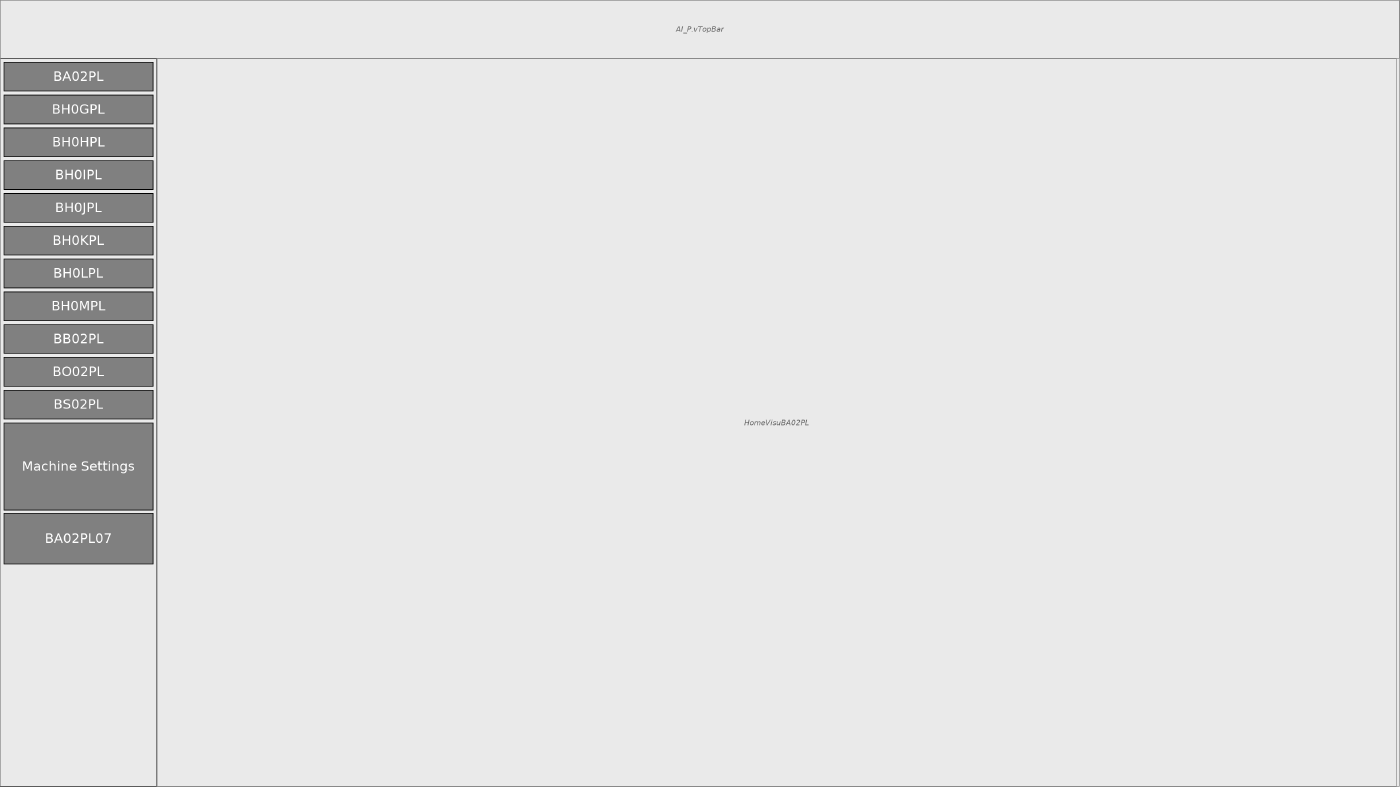
VISUALIZATION HomeVisu_1  // 1920x1080
    Rectangle (0,80 215x1000)
    Frame (215,80 1700x1000)
        shows HomeVisuBA02PL()
        shows HomeVisuBH0GPL()
        shows HomeVisuBH0HPL()
        shows HomeVisuBH0IPL()
        shows HomeVisuBH0JPL()
        shows HomeVisuBH0KPL()
        shows HomeVisuBH0LPL()
        shows HomeVisuBH0MPL()
        shows HomeVisuBB02PL()
        shows HomeVisuBO02PL()
        shows HomeVisuBS02PL()
        shows vHotPlateSettings_V3_B02PL(fbHP1_M1 := MAIN.fbHotPlate_G1_M1, fbHP1_M2 := MAIN.fbHotPlate_G1_M2, fbHP1_M3 := MAIN.fbHotPlate_G1_M3, fbHP2_M1 := MAIN.fbHotPlate_G2_M1, fbHP2_M2 := MAIN.fbHotPlate_G2_M2, fbHP2_M3 := MAIN.fbHotPlate_G2_M3, fbHP3_M1 := MAIN.fbHotPlate_G3_M1, fbHP3_M2 := MAIN.fbHotPlate_G3_M2, fbHP3_M3 := MAIN.fbHotPlate_G3_M3, fbHP4_M1 := MAIN.fbHotPlate_G4_M1, fbHP4_M2 := MAIN.fbHotPlate_G4_M2, fbHP4_M3 := MAIN.fbHotPlate_G4_M3, fbHP5_M1 := MAIN.fbHotPlate_G5_M1, fbHP5_M2 := MAIN.fbHotPlate_G5_M2, fbHP5_M3 := MAIN.fbHotPlate_G5_M3, fbHP6_M1 := MAIN.fbHotPlate_G6_M1, fbHP6_M2 := MAIN.fbHotPlate_G6_M2, fbHP6_M3 := MAIN.fbHotPlate_G6_M3, fbHP7_M1 := MAIN.fbHotPlate_G7_M1, fbHP7_M2 := MAIN.fbHotPlate_G7_M2, fbHP7_M3 := MAIN.fbHotPlate_G7_M3, fbS01_Press := MAIN.fbS01_BearingPress, fbS01_FixtureBase := MAIN.fbS01_KeyencePNVisSens, fbS02_Press := MAIN.fbS02_BearingPress, fbS03_Press := MAIN.fbS03_BearingPress, fbS03_FixtureBase := MAIN.fbS03_CapFixture, fbS04_Press := MAIN.fbS04_BearingPress, stHMIData_Filler_A := MAIN.fb_Filler_A_Machine.stHMI, stParams_Filler_A := MAIN.fb_Filler_A_Machine.stSlaveParms, stHMIData_Cork := MAIN.fb_Cork_Machine.stHMI, stParams_Cork := MAIN.fb_Cork_Machine.stSlaveParms, stHMIData_Filler_B := MAIN.fb_Filler_B_Machine.stHMI, stParams_Filler_B := MAIN.fb_Filler_B_Machine.stSlaveParms, stHMIData_Sticker := MAIN.fb_Sticker_Machine.stHMI, stParams_Sticker := MAIN.fb_Sticker_Machine.stSlaveParms, stHMIData_Laser := MAIN.fb_Laser_Machine.stHMI, stParams_Laser := MAIN.fb_Laser_Machine.stSlaveParms, stHMI_Laser := MAIN.fb_Laser_Machine.fbLaserControl.stHMI_Laser, fbSonic_S02 := MAIN.fb_1_SonicTech_SonictechUSW, fbSonic_S04 := MAIN.fb_2_SonicTech_SonictechUSW, fbVacuumChamber := MAIN.fb_UnderPressure_Tester_Machine, fbTransporter := MAIN.fbTransporterUnderpressure)
        shows AI_M.vWeighingTunnel(fbWeighingTunel := MAIN.fbWeighingTunel)
        shows vWeighingTunelVisionFrame()
        shows vStations19_21_22()
        p3043078949: MAIN.fbLL19_1_EOL3
        p1709583229: GVL.stLL19_EOL_Settings_I
        p2719655782: MAIN.fbLL19_2_EOL3
        p3094409976: GVL.stLL19_EOL_Settings_II
        p74549115: 'Left chamber'
        p3369830373: 'Right chamber'
        p4001053958: MAIN.fbS21_DetectionTunel
        p3623223747: MAIN.fbS21_DetectionTunel
        p3171485557: GVL.stS21_DTL_WorkParams
        p817651737: MAIN.stStation_LCA01PL_SCA01PL21
        p3449029454: GVL.stS21_DTL_Settings
        p3777340465: MAIN.fbS19_RecipeManager
        p3453682166: MAIN.stS19_EOL3_TMP_TestParams
        p3169997168: GVL_IO.stS21_DTL_InOuts.iLaserCurrentValue
        p2878062980: MAIN.fbS11_ResWelder.fbPIM
        p847417406: MAIN.fbS12_HiosScrewDriver.fbPIM
        p1166385320: MAIN.fbS13_FrontFanPress.fbPIM
        p3688969483: MAIN.fbS14_AssemblyPostCtrl.fbPIM
        p2900755869: MAIN.fbS15_AssemblyPostCtrl.fbPIM
        p3528948000: MAIN.fbS18_LabelSticking.fbPIM
        p514386723: MAIN.fbS22_SetPackingStation
        p2740858475: MAIN.fbS18_LabelSticking.stInOuts.iPressure
        p901175331: MAIN.fbS18_LabelSticking.stTestParams
        p1258792094: MAIN.fbS15_AssemblyPostCtrl.stWorkParams
        p1006670856: MAIN.fbS14_AssemblyPostCtrl.stWorkParams
        p2724463019: MAIN.fbS13_FrontFanPress.stParams
        p3580047677: MAIN.fbS12_HiosScrewDriver.stTestParam
        p1282039943: MAIN.fbS11_ResWelder.stWorkParams
        p285620971: GVL.stS19_EOL_TestParams
        p2487237938: MAIN.fbS19_1_EOL3
        p1850671185: MAIN.fbS19_2_EOL3
        p4100169850: GVL.stS19_EOL_Settings_I
        p241999129: GVL.stS19_EOL_Settings_II
        p1128139719: MAIN.fbS11_ResWelder.fbPIM
        p3661060733: MAIN.fbS12_HiosScrewDriver.fbPIM
        p2905631467: MAIN.fbS13_FrontFanPress.fbPIM
        p861208392: MAIN.fbS14_AssemblyPostCtrl.fbPIM
        p1146343390: MAIN.fbS15_AssemblyPostCtrl.fbPIM
        p987935587: MAIN.fbS18_LabelSticking.fbPIM
        p3446969237: GVL.stS18_ManometerCalibration_TestData
        p715956300: GVL.stS18_PressureScalingData
        p3016093480: GVL.stS15_AssemblyPostParams
        p3301105598: GVL.stS14_AssemblyPostParams
        p1520847389: GVL.stS13_Parameters
        p765557387: GVL.stS12_Parameters
        p3030919985: MAIN.fbS11_ResWelder.stWorkParams
        p4053094083: MAIN.fbS22_SetPackingStation
        p662549438: MAIN.fbS18_LabelSticking.stInOuts.iPressure
        p2928623001: GVL.stS18_PressureScalingData
        p1931357957: MAIN.fbS01_SonictechUSW.fbPIM
        p2635091497: MAIN.fbS03_SonictechUSW.fbPIM
        p1953753884: MAIN.fbS05_1_SonictechUSW.fbPIM
        p3984243366: MAIN.fbS06_SonictechUSW.fbPIM
        p2591918640: MAIN.fbS07_SonictechUSW.fbPIM
        p180524961: MAIN.fbS08_SonictechUSW.fbPIM
        p2110105399: MAIN.fbS09_SonictechUSW.fbPIM
        p486682322: MAIN.fbS10_SonictechUSW.fbPIM
        p4100033511: MAIN.fbS16_SonictechUSW.fbPIM
        p2204547953: MAIN.fbS17_SonictechUSW.fbPIM
        p3358502448: MAIN.fbS07_FixCarrierPistonAssy.stInOuts.rHeatStampTemperature
        p3363745968: GVL.stS01_FixSettings
        p644927900: GVL.stS03_FixSettings
        p3474158761: GVL.stS05_BallPressSettings
        p2347394456: GVL.stS05_USWelderSettings
        p1444554003: GVL.stS06_FixSettings
        p555554181: GVL.stS07_FixSettings
        p2980186132: GVL.stS08_FixSettings
        p3332716674: GVL.stS09_USWelderSettings
        p2791485799: GVL.stS10_USWelderSettings
        p1325470802: GVL.stS16_FixSettings
        p939926724: GVL.stS17_FixSettings
        p2967930134: GVL.stS21_DTL_Settings
        p2380948999: GVL_IO.stS21_DTL_InOuts.iLaserCurrentValue
        p3200496103: MAIN.fb_UnderPressure_Tester_Machine.stInOuts
        p980272329: MAIN.fb_UnderPressure_Tester_Machine.stParams
        p182610665: MAIN.fb_UnderPressure_Tester_Machine.stStatus
        p3000099066: MAIN.fb_UnderPressure_Tester_Machine.iWorkStep
        p1064606418: MAIN.fbTransporterUnderpressure.stInOuts
        p3808140917: MAIN.fbTransporterUnderpressure.stStatus
        p1825866306: MAIN.fbTransporterUnderpressure.iWorkStep
    Frame (0,0 1920x80)
        shows AI_P.vTopBar(fbLine := MAIN.stLine_BA02PL.fbLine)
    Rectangle (5,85 205x40), "BA02PL"
        OnMouseDown: FrameSelectionChange Selection=SelectedFrame=6c9ea511-e956-4d78-8ee8-89cc4cfbd0e1, GlobSel=AssignType=Directly, SelType=Locally
    Rectangle (5,130 205x40), "BH0GPL"
        OnMouseDown: FrameSelectionChange Selection=SelectedFrame=6c9ea511-e956-4d78-8ee8-89cc4cfbd0e1, Selection=1, GlobSel=AssignType=Directly, SelType=Locally
    Rectangle (5,580 205x120), "Machine Settings"
        OnMouseDown: FrameSelectionChange Selection=SelectedFrame=6c9ea511-e956-4d78-8ee8-89cc4cfbd0e1, Selection=11, GlobSel=AssignType=Directly, SelType=Locally
    Rectangle (5,175 205x40), "BH0HPL"
        OnMouseDown: FrameSelectionChange Selection=SelectedFrame=6c9ea511-e956-4d78-8ee8-89cc4cfbd0e1, Selection=2, GlobSel=AssignType=Directly, SelType=Locally
    Rectangle (5,265 205x40), "BH0JPL"
        OnMouseDown: FrameSelectionChange Selection=SelectedFrame=6c9ea511-e956-4d78-8ee8-89cc4cfbd0e1, Selection=4, GlobSel=AssignType=Directly, SelType=Locally
    Rectangle (5,220 205x40), "BH0IPL"
        OnMouseDown: FrameSelectionChange Selection=SelectedFrame=6c9ea511-e956-4d78-8ee8-89cc4cfbd0e1, Selection=3, GlobSel=AssignType=Directly, SelType=Locally
    Rectangle (5,310 205x40), "BH0KPL"
        OnMouseDown: FrameSelectionChange Selection=SelectedFrame=6c9ea511-e956-4d78-8ee8-89cc4cfbd0e1, Selection=5, GlobSel=AssignType=Directly, SelType=Locally
    Rectangle (5,355 205x40), "BH0LPL"
        OnMouseDown: FrameSelectionChange Selection=SelectedFrame=6c9ea511-e956-4d78-8ee8-89cc4cfbd0e1, Selection=6, GlobSel=AssignType=Directly, SelType=Locally
    Rectangle (5,445 205x40), "BB02PL"
        OnMouseDown: FrameSelectionChange Selection=SelectedFrame=6c9ea511-e956-4d78-8ee8-89cc4cfbd0e1, Selection=8, GlobSel=AssignType=Directly, SelType=Locally
    Rectangle (5,400 205x40), "BH0MPL"
        OnMouseDown: FrameSelectionChange Selection=SelectedFrame=6c9ea511-e956-4d78-8ee8-89cc4cfbd0e1, Selection=7, GlobSel=AssignType=Directly, SelType=Locally
    Rectangle (5,490 205x40), "BO02PL"
        OnMouseDown: FrameSelectionChange Selection=SelectedFrame=6c9ea511-e956-4d78-8ee8-89cc4cfbd0e1, Selection=9, GlobSel=AssignType=Directly, SelType=Locally
    Rectangle (5,535 205x40), "BS02PL"
        OnMouseDown: FrameSelectionChange Selection=SelectedFrame=6c9ea511-e956-4d78-8ee8-89cc4cfbd0e1, Selection=10, GlobSel=AssignType=Directly, SelType=Locally
    Rectangle (5,704 205x70), "BA02PL07"
        OnMouseDown: FrameSelectionChange Selection=SelectedFrame=6c9ea511-e956-4d78-8ee8-89cc4cfbd0e1, Selection=12, GlobSel=AssignType=Directly, SelType=Locally
END_VISUALIZATION

(* stored: Version 1.1.0.1, ProductVersion 3.1.4024.16
   Visu HomeVisu_1: Id {93810907-1595-475d-87cc-ce1c53c00b5f} *)
